Fanuc KAREL source: kf00087.KL

-- PROVISIONAL review KL for V770-1; original PC SHA256 0eb164538f86e9dcda77d86513347138d4f5511534283c008f17b0ddc8af7b42
-- Incomplete behavior may be omitted. Consult companion uncertainty JSON. Do not deploy.
PROGRAM KF00087
%NOLOCKGROUP
BEGIN
  -- UNRESOLVED_PC offsets 5-28; opcodes 27,22,1C,31,4A
  -- UNRESOLVED_PC offsets 33-37; opcodes 7F
END KF00087
